// TIA Portal V15.1 export
// export: Created 2022-12-20T09:13:23.7339052Z, ExportSetting None, DisplayName Totally Integrated Automation Portal, DisplayVersion V15.1 Update 1, DisplayName TIA Portal Openness, DisplayVersion V15.1, DisplayName SINAMICS Startdrive Advanced, DisplayVersion V15.1, DisplayName G130, G150, S120, S150, SINAMICS MV, S210, DisplayVersion V15.1, DisplayName G110M, G120, G120C, G120D, G120P, DisplayVersion V15.1, DisplayName STEP 7 Professional, DisplayVersion V15.1 Update 1, DisplayName STEP 7 Safety, DisplayVersion V15.1, DisplayName WinCC Professional, DisplayVersion V15.1 Update 1, DisplayName SIMATIC Visualization Architect, DisplayVersion V15.1
FUNCTION_BLOCK "PLC_MISCELLANEOUS_FB"   // FB513, LAD
TITLE = PLC MISCELLANEOUS FB
{ S7_Optimized_Access := 'TRUE' }
// The block is used to control equipment that is not linked to one SA or EM
// stored: AutoNumber false, MemoryReserve 100, SetENOAutomatically False
   VAR
      "000-HIP-SP11" : "CM_Digital_Input_FB";   // Zone panel air present
      "000-400K2" : "CM_Relay_FB";   // ++000+400K2
      "000-400K10" : "CM_Relay_FB";   // ++000+400K10
   END_VAR
BEGIN

REGION Network 1: Settings 000-HIP-SP11
   // Settings are: 
   // - Alarm when not active
   // - Alarm level drop running
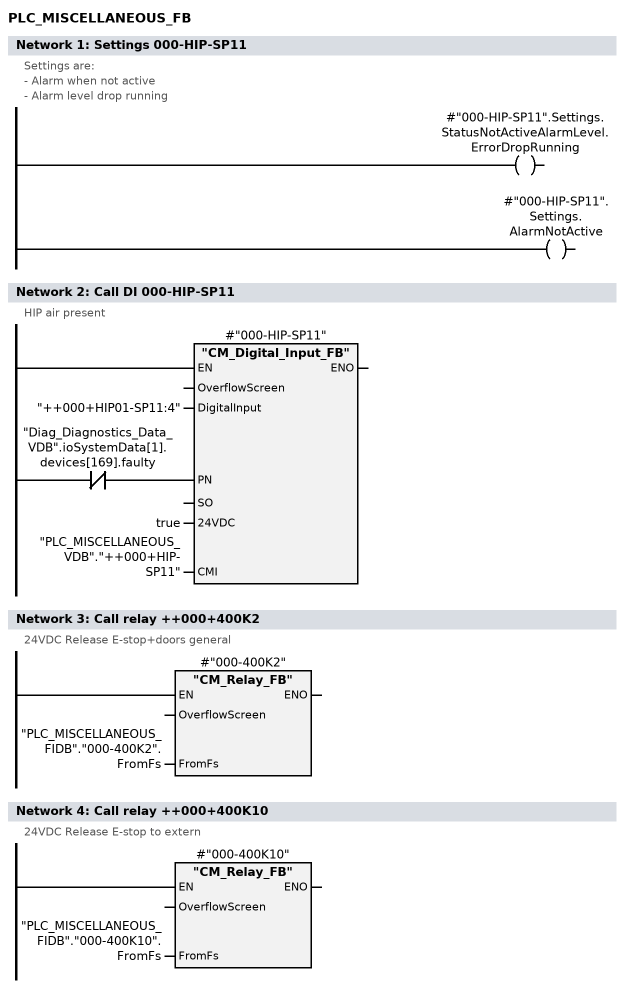
   RUNG wire#powerrail
      Coil( #"000-HIP-SP11".Settings.StatusNotActiveAlarmLevel.ErrorDropRunning )
   END_RUNG
   RUNG wire#powerrail
      Coil( #"000-HIP-SP11".Settings.AlarmNotActive )
   END_RUNG
   // the same network as SCL:
   #"000-HIP-SP11".Settings.StatusNotActiveAlarmLevel.ErrorDropRunning := TRUE;
   #"000-HIP-SP11".Settings.AlarmNotActive := TRUE;
END_REGION

REGION Network 2: Call DI 000-HIP-SP11
   // HIP air present
   RUNG wire#powerrail
      #"000-HIP-SP11"(PN := wire#w1, OverflowScreen :=, DigitalInput := "++000+HIP01-SP11:4", SO :=, "24VDC" := true, CMI := "PLC_MISCELLANEOUS_VDB"."++000+HIP-SP11")
   END_RUNG
   RUNG wire#powerrail
      I_Contact( "Diag_Diagnostics_Data_VDB".ioSystemData[1].devices[169].faulty )
   END_RUNG wire#w1
   // the same network as SCL:
   #"000-HIP-SP11"(DigitalInput := "++000+HIP01-SP11:4",   // "CM_Digital_Input_FB"
                   PN := NOT "Diag_Diagnostics_Data_VDB".ioSystemData[1].devices[169].faulty,
                   "24VDC" := true,
                   CMI := "PLC_MISCELLANEOUS_VDB"."++000+HIP-SP11");
END_REGION

REGION Network 3: Call relay ++000+400K2
   // 24VDC Release E-stop+doors general
   RUNG wire#powerrail
      #"000-400K2"(OverflowScreen :=, FromFs := "PLC_MISCELLANEOUS_FIDB"."000-400K2".FromFs)
   END_RUNG
   // the same network as SCL:
   #"000-400K2"(FromFs := "PLC_MISCELLANEOUS_FIDB"."000-400K2".FromFs);   // "CM_Relay_FB"
END_REGION

REGION Network 4: Call relay ++000+400K10
   // 24VDC Release E-stop to extern
   RUNG wire#powerrail
      #"000-400K10"(OverflowScreen :=, FromFs := "PLC_MISCELLANEOUS_FIDB"."000-400K10".FromFs)
   END_RUNG
   // the same network as SCL:
   #"000-400K10"(FromFs := "PLC_MISCELLANEOUS_FIDB"."000-400K10".FromFs);   // "CM_Relay_FB"
END_REGION
END_FUNCTION_BLOCK
